INTERFACE I_RegisterPosition

METHOD RegisterPosition : BOOL
VAR_INPUT
	position : I_Position;
END_VAR
END_METHOD

END_INTERFACE

(* stored: Version 1.1.0.1
   Itf I_RegisterPosition: Id {1e05ceef-0262-4a21-a758-47139e8aa10c}
   Method RegisterPosition: Id {8700400e-5434-4855-973a-1d39e7085e82} *)
